Staubli VAL3: sad_project_1.pjx

--- sad_project_1.pjx ---
Parameters version=s7.7.1 stackSize=5000 millimeterUnit=true
Program file=check_cmt.pgx
Program file=motion_cntl.pgx
Program file=open_socket.pgx
Program file=open_socket1.pgx
Program file=read_data.pgx
Program file=send_data.pgx
Program file=show_data.pgx
Program file=start.pgx
Program file=stop.pgx
Data file=sad_project_1.dtx

--- sad_project_1.dtx ---
public num Ref_Vel
public mdesc mNomSpeed = {tmax=100, rmax=100, leave=0.1, reach=0.1, blend=off}
public jointRx Jnt_cnfg = {j3=90, j5=90, j6=90}
public tool tTool = {z=600, rz=55, fatherId=flange[0], ioLink=valve1}
public frame fReference = {x=1365.054, y=-125.975, z=-1150, fatherId=world[0]}
public pointRx Pnt_1st_lyr[2]
  [0] = {y=-1000, rx=-180, rz=-90, shoulder=lefty, elbow=epositive, wrist=wpositive, fatherId=fReference[0]}
  [1] = {y=1000, rx=-180, rz=-90, shoulder=lefty, elbow=epositive, wrist=wpositive, fatherId=fReference[0]}
public pointRx Pnt_2nd_lyr[4]
  [0] = {y=1000, z=77, rx=180, rz=-90, shoulder=lefty, elbow=epositive, wrist=wpositive, fatherId=fReference[0]}
  [1] = {y=-1000, z=77, rx=180, rz=-90, shoulder=lefty, elbow=epositive, wrist=wpositive, fatherId=fReference[0]}
  [2] = {y=-1000, z=22, rx=180, rz=-90, shoulder=lefty, elbow=epositive, wrist=wpositive, fatherId=fReference[0]}
  [3] = {y=1000, z=22, rx=180, rz=-90, shoulder=lefty, elbow=epositive, wrist=wpositive, fatherId=fReference[0]}
public pointRx Pnt_3rd_lyr[4]
  [0] = {y=1000, z=99, rx=180, rz=-90, shoulder=lefty, elbow=epositive, wrist=wpositive, fatherId=fReference[0]}
  [1] = {y=-1000, z=99, rx=180, rz=-90, shoulder=lefty, elbow=epositive, wrist=wpositive, fatherId=fReference[0]}
  [2] = {y=-1000, z=44, rx=180, rz=-90, shoulder=lefty, elbow=epositive, wrist=wpositive, fatherId=fReference[0]}
  [3] = {y=1000, z=44, rx=180, rz=-90, shoulder=lefty, elbow=epositive, wrist=wpositive, fatherId=fReference[0]}
public pointRx Pnt_4th_lyr[4]
  [0] = {y=1000, z=116, rx=180, rz=-90, shoulder=lefty, elbow=epositive, wrist=wpositive, fatherId=fReference[0]}
  [1] = {y=-1000, z=116, rx=180, rz=-90, shoulder=lefty, elbow=epositive, wrist=wpositive, fatherId=fReference[0]}
  [2] = {y=-1000, z=66, rx=180, rz=-90, shoulder=lefty, elbow=epositive, wrist=wpositive, fatherId=fReference[0]}
  [3] = {y=1000, z=66, rx=180, rz=-90, shoulder=lefty, elbow=epositive, wrist=wpositive, fatherId=fReference[0]}
public trsf trTrsf
sio sioASCII = {link=Socket\trsf_sv}
public bool check_status
public bool spd_cntl
public mdesc cnst_vel = {tmax=100, rmax=100, leave=0.1, reach=0.1, blend=cartesian}
aio Tpompe = {link=CanIO\RemIO\remio0_QW}
dio doValve1 = {link=valve1}
dio doValve2 = {link=valve2}

--- open_socket.pgx ---
public program open_socket()
begin

  //sioCtrl(sioASCII,"port",11002)
  sioCtrl(sioASCII,"port",1002)
  //sioCtrl(sioASCII,"target","10.3.1.185")
  sioCtrl(sioASCII,"target","10.10.5.1")
  //sioCtrl(sioASCII,"target","169.254.209.1")
  sioCtrl(sioASCII,"timeout",10)
  sioCtrl(sioASCII,"endOfString",13)
  sioCtrl(sioASCII,"nangle",true)

  putln(" " )
  putln("The communication socket is open.")

  check_status = false

end

--- read_data.pgx ---
public program read_data()
  local string sInputData_1
  local num nRec
  local num nReceived
  local num nInputData_1
begin

  putln("Start to read data !")

  do
    sInputData_1 = ""
    do
      nReceived=sioGet(sioASCII,nRec)
      sInputData_1 = sInputData_1 + chr(nRec)

    until nRec == 13 or nReceived == -1

    if nReceived != 1
      check_status = false
      stopMove()
      cls()
      putln("Communication error !")
      disablePower()
    endIf

    toNum(sInputData_1 , nInputData_1, check_status)

    //put("Reference Velocity [mm/s]: ")
    //put(nInputData_1)
    //putln("")



    if getMoveId() >= 0.1
       Ref_Vel = nInputData_1
    elseIf getMoveId() < 0.1
       Ref_Vel = print_vel
    endIf

   // putln(Ref_Vel)


   //delay(0.001)

  until check_status != true

end

--- send_data.pgx ---
program send_data()
  local string snd_msg
  local num i
  local num nSent
begin

  putln("Start to send data !")

  do

  snd_msg = toString(".4",getSpeed(tTool)) + chr(13) + chr(10)

  for i=0 to len(snd_msg)-1
    nSent = sioSet(sioASCII,asc(snd_msg,i))

    if nSent != 1
      check_status = false
      stopMove()
      cls()
      putln("Communication error !")
      disablePower()
    endIf


  endFor

  //putln(snd_msg)

  //cls()
  delay(.2)

  until check_status != true


end

--- stop_print.pgx ---
public program stop_print()
begin

      // arrêt pompe
    dioSet(doPompe,0)
    put("Pompe arret")
      // fermeture obturateur
    dioSet(doValve2,0)
    dioSet(doValve1,1)
    put("Obturateur ferme")

end
